PROGRAM ControlMachine
VAR_input
	xAlarm                      	: BOOL;
	tonEmptyDone	: TON;					//Empty Done Delay
	bEmptyDone                  	: BOOL ;
	
	
END_VAR
VAR
	i,j : INT ;
	_xMaterialOnFlag : BOOL ;//环形线
	
	
	tTimeoutAlarm: TON;
	tCounterR_TRIG: R_TRIG;
	tCounter1R_TRIG: R_TRIG;
	tCounter2R_TRIG: R_TRIG;
	tPCAlarmR_TRIG: R_TRIG;
END_VAR

A_Input();
Safety();
Waiting();
Timeout();
Alarm();
CycleTime();
Tip();
InitDone();
EmptyDone();
General();
Z_Output();

ACTION A_Input:

END_ACTION

ACTION Alarm:
//----机台状态提示---//
fbMachine[1].dwMessage[1].00			:=	fbMachine[1].xRunning;			//设备自动中
fbMachine[1].dwMessage[1].01		    :=	fbMachine[1].xStopped;			//设备停止状态
fbMachine[1].dwMessage[1].02			:=	fbMachine[1].xPaused;			//设备暂停状态
fbMachine[1].dwMessage[1].03			:=	fbMachine[1].xAlarm;			//设备报警中
fbMachine[1].dwMessage[1].04			:=	fbMachine[1].xIniting;			//设备初始化中
fbMachine[1].dwMessage[1].05			:=	fbMachine[1].xEmptying;			//设备清料中

//----机台报警信息----
//IF NOT  fbMachine[1].xAirOn THEN
//	fbMachine[1].dwAlarm[1].00:=TRUE; //[M01.00] 设备气压报警
//	;
//END_IF
//急停被按下
IF NOT IxSafetyRelayOK THEN 
	fbMachine[1].dwAlarm[1].03:=TRUE; //[M01.03] 设备急停被按下
END_IF

//心跳
//	IF  fbAlive[1].xQAliveError THEN
//		fbMachine[1].dwAlarm[1].05:=TRUE; //[M01.05] 未检测到相机心跳1
//	END_IF
//	IF  fbAlive[2].xQAliveError THEN
//		fbMachine[1].dwAlarm[1].06:=TRUE; //[M01.06] 未检测到相机心跳2
//	END_IF
//	IF  fbAlive[3].xQAliveError THEN
//		fbMachine[1].dwAlarm[1].07:=TRUE; //[M01.07] 未检测到相机心跳3
//	END_IF
//	IF  fbAlive[4].xQAliveError THEN
//		fbMachine[1].dwAlarm[1].08:=TRUE; //[M01.08] 未检测到工控机1心跳
//	END_IF
//	IF  fbAlive[5].xQAliveError THEN
//		fbMachine[1].dwAlarm[1].09:=TRUE; //[M01.09] 未检测到工控机2心跳
//	END_IF
//	IF  fbAlive[6].xQAliveError THEN
//		fbMachine[1].dwAlarm[1].10:=TRUE; //[M01.10] 未检测到工控机3心跳
//	END_IF
//	IF  fbAlive[7].xQAliveError THEN
//		fbMachine[1].dwAlarm[1].11:=TRUE; //[M01.11] 未检测到热缩封膜机心跳
//	END_IF
////模块状态
//	IF  fbEhterCATSlaveMonitor[1].xQError THEN
//		fbMachine[1].dwAlarm[1].12:=TRUE; //[M01.05] ET01电柜EtherCAT总线报错
//	END_IF
//	IF  fbEhterCATSlaveMonitor[2].xQError THEN
//		fbMachine[1].dwAlarm[1].13:=TRUE; //[M01.05] ET02电柜EtherCAT总线报错
//	END_IF
//	IF  fbEhterCATSlaveMonitor[3].xQError THEN
//		fbMachine[1].dwAlarm[1].14:=TRUE; //[M01.05] ET03电柜EtherCAT总线报错
//	END_IF
//		IF  fbEhterCATSlaveMonitor[4].xQError THEN
//		fbMachine[1].dwAlarm[1].15:=TRUE; //[M01.05] ET04电柜EtherCAT总线报错
//	END_IF

	
	
//----工站报警汇总----

xAlarm:= FALSE;							//先复位
FOR i :=1 TO gc_uiStationNum DO 
  IF fbStation[i].xAlarm THEN		//整机故障单独 
    xAlarm:=TRUE; 
  END_IF
END_FOR

//----机台报警----
fbMachine[1].xAlarm:=
  fbMachine[1].dwAlarm[1]<>0
	OR fbMachine[1].dwAlarm[2]<>0
	OR fbMachine[1].dwAlarm[3]<>0
	OR fbMachine[1].dwAlarm[4]<>0
	OR fbMachine[1].dwAlarm[5]<>0
	OR xAlarm;
END_ACTION

ACTION CycleTime:
//**************************计算循环周期*******************************///
END_ACTION

ACTION EmptyDone:
(*
tonEmptyDone(
	IN:=fbMachine[1].xEmptying AND ( abClearMaterialOver[gc_uiStationNum] OR NOT _xMaterialOnFlag ) AND fbMachine[1].xRunning,
	PT:=T#2S,
	Q=>, ET=>
);

IF tonEmptyDone.Q THEN
   fbMachine[1].xEmptyDone:=TRUE;
   FOR i :=1 TO gc_uiStationNum DO 
	  abClearMaterialOver[i] :=FALSE;  
   END_FOR
   ////////////////工站间的交互信号处理或者其他信号///////////////////
END_IF
*)


//**********************设备有料标志位*********
_xMaterialOnFlag := FALSE ;
FOR i:=1 TO 40 BY 1 DO 
 IF arMainlineFixtureData[i].xMaterialOnOff  THEN 
	  _xMaterialOnFlag := TRUE ;
 END_IF
END_FOR
END_ACTION

ACTION General:

//设备总产量
  fbMachine[1].udiTotal := fbMachine[1].udiGoods + fbMachine[1].udiBads ;

//产量清除
  IF fbMachine[1].xClearCountData THEN 
	  fbMachine[1].udiGoods := fbMachine[1].udiBads := 0 ;
	  fbMachine[1].xClearCountData:=FALSE;
  END_IF
  
//产品计数
(*
tCounterR_TRIG(CLK:=S07_Unloading.xBothPartGoodFlag, Q=> );
tCounter1R_TRIG(CLK:=S07_Unloading.xOnePartGoodFlag , Q=> );
tCounter2R_TRIG(CLK:=S07_Unloading.xOnePartBadFlag , Q=> );
*)
IF  tCounterR_TRIG.Q THEN
	fbMachine[1].udiGoods := fbMachine[1].udiGoods + 2;	//设备OK产品计数
ELSIF  tCounter1R_TRIG.Q  THEN
	fbMachine[1].udiGoods := fbMachine[1].udiGoods + 1;	//设备OK产品计数
ELSIF  tCounter2R_TRIG.Q THEN
	fbMachine[1].udiBads := fbMachine[1].udiBads + 1;	//设备OK产品计数	
END_IF
END_ACTION

ACTION InitDone:

//------------------------------------------------初始化完成汇总-------------------------------------

fbMachine[1].xInitDone:=TRUE;//先置位
FOR j :=1 TO gc_uiStationNum DO 
  IF NOT fbStation[j].xInitDone
  THEN 
    fbMachine[1].xInitDone:=FALSE; 
  END_IF
END_FOR
END_ACTION

ACTION Safety:
//-------------------------------------------------安全信号------------------------------------------------------

//fbMachine[1].xDoorClosed:= fbSafetyDoor[1].xLocked ;
						
//fbSafetyDoor[1].xUnlock:= FALSE;
fbMachine[1].xDoorClosed := TRUE ;

fbMachine[1].xEStop :=IxSafetyRelayOK ;					   

fbMachine[1].xKey := TRUE;

fbMachine[1].xAirOn :=  IxAirPressure OR true;

fbMachine[1].xSafety:=fbMachine[1].xDoorClosed 
						AND fbMachine[1].xEStop 
						AND fbMachine[1].xAirOn 
						AND fbMachine[1].xKey ;
END_ACTION

ACTION Timeout:

END_ACTION

ACTION Tip:
//------------------------------------------------提示汇总-----------------------------------------------
//----手动提示----
fbMachine[1].xManualTip                :=FALSE;//先复位
FOR j:=1 TO gc_uiStationNum DO 
  IF fbStation[j].xManualTip THEN 
   fbMachine[1].xManualTip            :=TRUE; 
  END_IF
END_FOR

//----自动提示----
fbMachine[1].xAutoTip                  :=FALSE;//先复位
FOR j :=1 TO gc_uiStationNum DO 
  IF fbStation[j].xAutoTip
  THEN 
   fbMachine[1].xAutoTip              :=TRUE; 
  END_IF
END_FOR

fbMachine[1].xTip                      :=(fbMachine[1].xManualTip OR fbMachine[1].xAutoTip);
/////////////////////////////////////////////////////////////////////////////////////////////////////////
END_ACTION

ACTION Waiting:

END_ACTION

ACTION Z_Output:

END_ACTION

END_PROGRAM

(* stored: Version 1.1.0.1, ProductVersion 3.1.4024.9
   POU ControlMachine: Id {c5f22d68-fa5f-404d-9f0e-4fab1cd07031}, SpecialFunc None
   Action A_Input: Id {0714662c-3b58-40cf-a1d8-1883f3374852}
   Action Alarm: Id {040003db-0126-4202-b8aa-167197bcc773}
   Action CycleTime: Id {f5fed5cc-8ba8-475b-ad40-4130d1b07351}
   Action EmptyDone: Id {2aec48a2-7e6f-44b6-b88a-567108dc02b2}
   Action General: Id {59fdc1bd-eac6-41d6-8b9d-30b7eb5e0166}
   Action InitDone: Id {4d14d86d-8273-43c8-916f-3a4bda99cb3c}
   Action Safety: Id {7756a730-2991-421a-83ea-4ae6ba5ac083}
   Action Timeout: Id {21e89cc2-bcd2-45fb-a2b6-ed65b1837306}
   Action Tip: Id {25a2cd35-9d8c-457b-9db7-ff9dd12f040c}
   Action Waiting: Id {ba3e6eab-3f00-42c5-91c9-b2be4453d15d}
   Action Z_Output: Id {99e18fa8-8f26-440f-bf00-acd6707ee93a} *)
